// TIA Portal project "MODBUS-2" (V17)

(* hardware
DEVICE "S7-1200 station_1"  S7-1200 Station
   slot 0: "Rack_0"  S7-1200 Rack  Rack  V1.0
   slot 1: "PLC_1"  CPU 1211C DC/DC/DC  6ES7 211-1AE40-0XB0  V4.5
*)

// ===== PLC "PLC_1"  CPU 1211C DC/DC/DC =====

VAR_GLOBAL   // PLC tag table "Default tag table"
   "System_Byte" AT %MB1 : Byte;
   "FirstScan" AT %M1.0 : Bool;
   "DiagStatusUpdate" AT %M1.1 : Bool;
   "AlwaysTRUE" AT %M1.2 : Bool;
   "AlwaysFALSE" AT %M1.3 : Bool;
   "Clock_Byte" AT %MB0 : Byte;
   "Clock_10Hz" AT %M0.0 : Bool;
   "Clock_5Hz" AT %M0.1 : Bool;
   "Clock_2.5Hz" AT %M0.2 : Bool;
   "Clock_2Hz" AT %M0.3 : Bool;
   "Clock_1.25Hz" AT %M0.4 : Bool;
   "Clock_1Hz" AT %M0.5 : Bool;
   "Clock_0.625Hz" AT %M0.6 : Bool;
   "Clock_0.5Hz" AT %M0.7 : Bool;
   "POWER ON" AT %M2.0 : Bool;
   "POWER READ" AT %M2.1 : Bool;
   "POWER WRITE" AT %M2.2 : Bool;
   "START-RD" AT %M2.3 : Bool;
   "START-WR" AT %M2.4 : Bool;
   "TIMEIN-RD" AT %MD4 : Time;
   "TIMEIN-WR" AT %MD8 : Time;
   "OUT-RD" AT %M2.5 : Bool;
   "TIMEOUT-RD" AT %MD12 : Time;
   "OUT-WR" AT %M2.6 : Bool;
   "TIMEOUT-WR" AT %MD16 : Time;
END_VAR

DATA_BLOCK "Data_block_RD"   // DB2
{ S7_Optimized_Access := 'FALSE' }
VERSION : 0.1
   VAR
      CONNECT : TCON_IP_v4;
      DISCONNECT : Bool;
      MODE : USInt := 0;
      DATA_ADDR : UDInt := 1;
      MB_DATA_LEN : UInt := 10;
      DONE : Bool;
      BUSY : Bool;
      ERROR : Bool;
      STATUS : Word;
   END_VAR
BEGIN
   CONNECT.InterfaceId := 64;
   CONNECT.ID := 3;
   CONNECT.ConnectionType := 11;
   CONNECT.ActiveEstablished := TRUE;
   CONNECT.RemotePort := 502;
   CONNECT.RemoteAddress.ADDR[4] := 177;
   CONNECT.RemoteAddress.ADDR[3] := 2;
   CONNECT.RemoteAddress.ADDR[2] := 168;
   CONNECT.RemoteAddress.ADDR[1] := 192;
END_DATA_BLOCK

DATA_BLOCK "SALIDAS"   // DB3
{ S7_Optimized_Access := 'FALSE' }
VERSION : 0.1
   VAR
      DATA_0 : Int;
      DATA_1 : Int;
      DATA_2 : Int;
      DATA_3 : Int;
      DATA_4 : Int;
      DATA_5 : Int;
      DATA_6 : Int;
      DATA_7 : Int;
      DATA_8 : Int;
      DATA_9 : Int;
   END_VAR
BEGIN
END_DATA_BLOCK

DATA_BLOCK "Data_block_WR"   // DB4
{ S7_Optimized_Access := 'FALSE' }
VERSION : 0.1
   VAR
      CONNECT : TCON_IP_v4;
      DISCONNECT : Bool;
      MODE : USInt := 1;
      DATA_ADDR : UDInt := 1;
      MB_DATA_LEN : UInt := 10;
      DONE : Bool;
      BUSY : Bool;
      ERROR : Bool;
      STATUS : Word;
   END_VAR
BEGIN
   CONNECT.InterfaceId := 64;
   CONNECT.ID := 3;
   CONNECT.ConnectionType := 11;
   CONNECT.ActiveEstablished := TRUE;
   CONNECT.RemotePort := 502;
   CONNECT.RemoteAddress.ADDR[4] := 177;
   CONNECT.RemoteAddress.ADDR[3] := 2;
   CONNECT.RemoteAddress.ADDR[2] := 168;
   CONNECT.RemoteAddress.ADDR[1] := 192;
END_DATA_BLOCK

// folder: System blocks/Program resources

DATA_BLOCK "TIMER-READ"   // DB5
{ S7_Optimized_Access := 'TRUE' }
AUTHOR : Simatic
FAMILY : IEC
NAME : IEC_TMR
VERSION : 1.0
// stored: InstanceOfName IEC_TIMER
"IEC_TIMER"
BEGIN
END_DATA_BLOCK

DATA_BLOCK "TIMER-WRITE"   // DB6
{ S7_Optimized_Access := 'TRUE' }
AUTHOR : Simatic
FAMILY : IEC
NAME : IEC_TMR
VERSION : 1.0
// stored: InstanceOfName IEC_TIMER
"IEC_TIMER"
BEGIN
END_DATA_BLOCK

// folder: (top level)

FUNCTION "FC-READ-WRITE" : Void   // FC1, LAD
{ S7_Optimized_Access := 'TRUE' }
VERSION : 0.1
BEGIN

REGION Network 1: READ
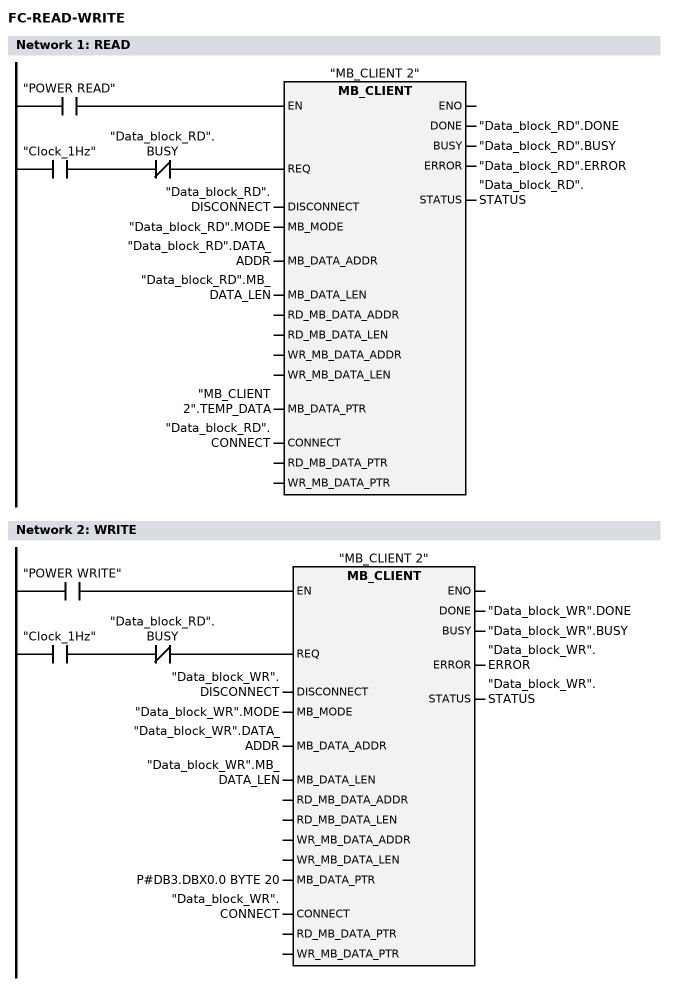
   IF "POWER READ" THEN
       "MB_CLIENT 2"(REQ := "Clock_1Hz" AND NOT "Data_block_RD".BUSY,   // MB_CLIENT
                     DISCONNECT := "Data_block_RD".DISCONNECT,
                     MB_MODE := "Data_block_RD".MODE,
                     MB_DATA_ADDR := "Data_block_RD".DATA_ADDR,
                     MB_DATA_LEN := "Data_block_RD".MB_DATA_LEN,
                     MB_DATA_PTR := "MB_CLIENT 2".TEMP_DATA,
                     CONNECT := "Data_block_RD".CONNECT,
                     DONE => "Data_block_RD".DONE,
                     BUSY => "Data_block_RD".BUSY,
                     ERROR => "Data_block_RD".ERROR,
                     STATUS => "Data_block_RD".STATUS);
   END_IF;
END_REGION

REGION Network 2: WRITE
   IF "POWER WRITE" THEN
       "MB_CLIENT 2"(REQ := "Clock_1Hz" AND NOT "Data_block_RD".BUSY,   // MB_CLIENT
                     DISCONNECT := "Data_block_WR".DISCONNECT,
                     MB_MODE := "Data_block_WR".MODE,
                     MB_DATA_ADDR := "Data_block_WR".DATA_ADDR,
                     MB_DATA_LEN := "Data_block_WR".MB_DATA_LEN,
                     MB_DATA_PTR := P#DB3.DBX0.0 BYTE 20,
                     CONNECT := "Data_block_WR".CONNECT,
                     DONE => "Data_block_WR".DONE,
                     BUSY => "Data_block_WR".BUSY,
                     ERROR => "Data_block_WR".ERROR,
                     STATUS => "Data_block_WR".STATUS);
   END_IF;
END_REGION

REGION Network 3 (SCL): SCL
   WHILE "POWER ON" = 1 DO
       IF "POWER READ" = 0 AND "POWER WRITE" = 0 THEN
           "POWER READ" := 1;
           "START-RD" := 1;
       END_IF;
       IF "POWER READ" = 1 AND "OUT-RD" = 1 THEN
           "POWER READ" := 0;
           "START-RD" := 0;
           "POWER WRITE" := 1;
           "START-WR" := 1;
       END_IF;
       IF "POWER WRITE" = 1 AND "OUT-WR" = 1 THEN
           "POWER WRITE" := 0;
           "START-WR" := 0;
       END_IF;
   END_WHILE;
END_REGION
END_FUNCTION

FUNCTION "FC-SCL-TIMERS" : Void   // FC3, SCL
{ S7_Optimized_Access := 'TRUE' }
VERSION : 0.1
   VAR_INPUT
      "START-RD" : Bool;
      "TIMEIN-RD" : Time;
      "START-WR" : Bool;
      "TIMEIN-WR" : Time;
   END_VAR
   VAR_OUTPUT
      "OUT-RD" : Bool;
      "TIMEOUT-RD" : Time;
      "OUT-WR" : Bool;
      "TIMEOUT-WR" : Time;
   END_VAR
BEGIN
   "TIMER-READ".TON(IN:=#"START-RD"=1,
                    PT:=#"TIMEIN-RD",
                    Q=>#"OUT-RD",
                    ET=>#"TIMEOUT-RD");
   "TIMER-WRITE".TON(IN:=#"START-WR"=1,
                     PT:=#"TIMEIN-WR",
                     Q=>#"OUT-WR",
                     ET=>#"TIMEOUT-WR");
END_FUNCTION

ORGANIZATION_BLOCK "Main"   // OB1, LAD, ProgramCycle
TITLE = "Main Program Sweep (Cycle)"
{ S7_Optimized_Access := 'TRUE' }
VERSION : 0.1
   VAR_INPUT
      Initial_Call : Bool;   // Initial call of this OB
      Remanence : Bool;   // =True, if remanent data are available
   END_VAR
BEGIN

REGION Network 1: POWER-ON
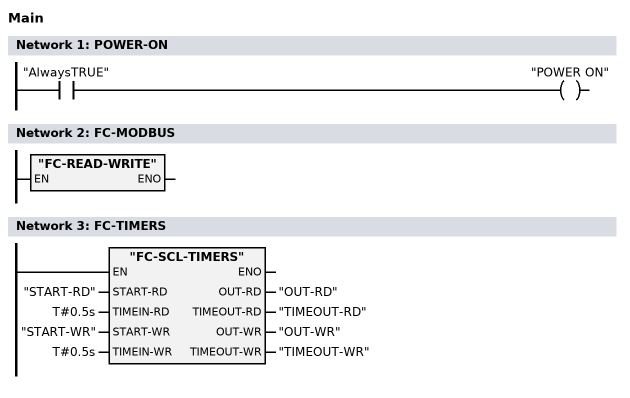
   RUNG wire#powerrail
      Contact( "AlwaysTRUE" )
      Coil( "POWER ON" )
   END_RUNG
   // the same network as SCL:
   "POWER ON" := "AlwaysTRUE";
END_REGION

REGION Network 2: FC-MODBUS
   RUNG wire#powerrail
      "FC-READ-WRITE"()
   END_RUNG
   // the same network as SCL:
   "FC-READ-WRITE"();
END_REGION

REGION Network 3: FC-TIMERS
   RUNG wire#powerrail
      "FC-SCL-TIMERS"("START-RD" := "START-RD", "TIMEIN-RD" := T#0.5s, "START-WR" := "START-WR", "TIMEIN-WR" := T#0.5s, "OUT-RD" => "OUT-RD", "TIMEOUT-RD" => "TIMEOUT-RD", "OUT-WR" => "OUT-WR", "TIMEOUT-WR" => "TIMEOUT-WR")
   END_RUNG
   // the same network as SCL:
   "FC-SCL-TIMERS"("START-RD" := "START-RD",
                   "TIMEIN-RD" := T#0.5s,
                   "START-WR" := "START-WR",
                   "TIMEIN-WR" := T#0.5s,
                   "OUT-RD" => "OUT-RD",
                   "TIMEOUT-RD" => "TIMEOUT-RD",
                   "OUT-WR" => "OUT-WR",
                   "TIMEOUT-WR" => "TIMEOUT-WR");
END_REGION
END_ORGANIZATION_BLOCK